// TIA Portal V16 export
// export: Created 2020-03-07T17:54:43.9298204Z, ExportSetting WithDefaults, DisplayName Totally Integrated Automation Portal, DisplayVersion V16 Update 1, DisplayName TIA Portal Version Control Interface, DisplayVersion V16, DisplayName TIA Portal Openness, DisplayVersion V16 Update 1, DisplayName STEP 7 Professional, DisplayVersion V16 Update 1, DisplayName STEP 7 Safety, DisplayVersion V16, DisplayName WinCC Professional, DisplayVersion V16 Update 1
ORGANIZATION_BLOCK "Main"   // OB1, LAD, ProgramCycle
TITLE = "Main Program Sweep (Cycle)"
{ S7_Optimized_Access := 'TRUE' }
VERSION : 0.1
// stored: AutoNumber true, IsIECCheckEnabled false, SetENOAutomatically false
   VAR_INPUT
      Initial_Call : Bool;   // Initial call of this OB
      Remanence : Bool;   // =True, if remanent data are available
   END_VAR
BEGIN

REGION Network 1
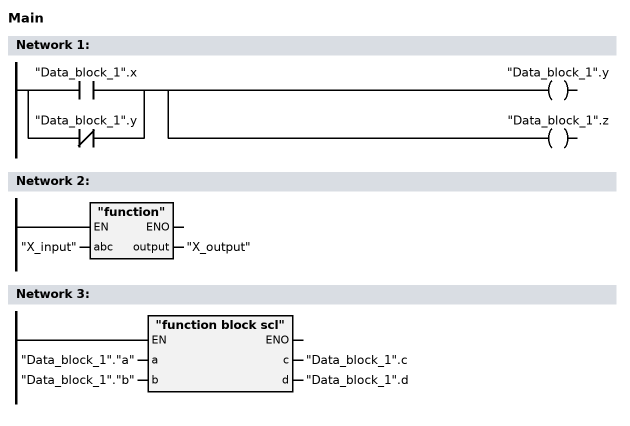
   RUNG wire#powerrail
      Contact( "Data_block_1".x )
      wire#w1
      Coil( "Data_block_1".y )
   END_RUNG
   RUNG wire#powerrail
      I_Contact( "Data_block_1".y )
   END_RUNG wire#w1
   RUNG wire#w1
      Coil( "Data_block_1".z )
   END_RUNG
   // the same network as SCL:
   "Data_block_1".y := "Data_block_1".x OR NOT "Data_block_1".y;
   "Data_block_1".z := "Data_block_1".y;
END_REGION

REGION Network 2
   RUNG wire#powerrail
      "function"(abc := "X_input", output => "X_output")
   END_RUNG
   // the same network as SCL:
   "function"(abc := "X_input", output => "X_output");
END_REGION

REGION Network 3
   RUNG wire#powerrail
      "function block scl"("a" := "Data_block_1"."a", "b" := "Data_block_1"."b", c => "Data_block_1".c, d => "Data_block_1".d)
   END_RUNG
   // the same network as SCL:
   "function block scl"("a" := "Data_block_1"."a",
                        "b" := "Data_block_1"."b",
                        c => "Data_block_1".c,
                        d => "Data_block_1".d);
END_REGION
END_ORGANIZATION_BLOCK
